// TIA Portal V18 export
DATA_BLOCK "L1_taglioValvProp"   // DB13
{ S7_Optimized_Access := 'TRUE' }
VERSION : 0.1
// stored: AutoNumber false, DBAccessibleFromOPCUA true, DBAccessibleFromWebserver true, IsOnlyStoredInLoadMemory false, IsRetainMemResEnabled false, IsWriteProtectedInAS false, MemoryReserve 100
   VAR RETAIN
      data : "LGasp_taglioValvProp";
      prg { ExternalAccessible := 'False'; ExternalVisible := 'False'; ExternalWritable := 'False'} : Array[1.."N_PrgValvole"] of "LGasp_taglioValvProp";
   END_VAR
BEGIN
END_DATA_BLOCK
